// LS Electric XG5000 project: xg1006
// PLC LSPLC
// module base 0 slot 0: 입력 모듈:XGI-D24A/B (DC 24V 입력, 32점 (전류소스 싱크공용/ 전류소스 입력))
// module base 0 slot 1: 출력 모듈:XGQ-TR4A/B (트랜지스터 출력, 32점 (0.1A용, 싱크출력/소스출력))

PROGRAM NewProgram (task: 스캔 프로그램)

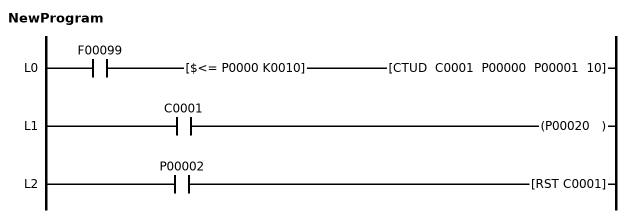
; L0
LOAD      F00099
AND$<=    P0000 K0010
CTUD      C0001 P00000 P00001 10
; L1
LOAD      C0001
OUT       P00020
; L2
LOAD      P00002
RST       C0001